FUNCTION_BLOCK SERVER_5 (* 5 SD/RD Server Interface *)
  (* Standard: 61499-1; Classification: Communications *)
  (* Version 0.0, 2004-04-29, JHC, Rockwell Automation *)
  (* Compiler header: package fb.rt.net; *)
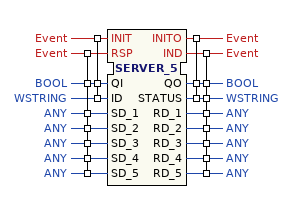
  EVENT_INPUT
    INIT WITH QI, ID;
    RSP WITH QI, SD_1, SD_2, SD_3, SD_4, SD_5;
  END_EVENT
  EVENT_OUTPUT
    INITO WITH QO, STATUS;
    IND WITH QO, STATUS, RD_1, RD_2, RD_3, RD_4, RD_5;
  END_EVENT
  VAR_INPUT
    QI : BOOL;
    ID : WSTRING;
    SD_1 : ANY;
    SD_2 : ANY;
    SD_3 : ANY;
    SD_4 : ANY;
    SD_5 : ANY;
  END_VAR
  VAR_OUTPUT
    QO : BOOL;
    STATUS : WSTRING;
    RD_1 : ANY;
    RD_2 : ANY;
    RD_3 : ANY;
    RD_4 : ANY;
    RD_5 : ANY;
  END_VAR
END_FUNCTION_BLOCK
